FUNCTION FUNC_Bad : BOOL
VAR_INPUT
  nInput : INT;
END_VAR

FUNC_Bad := nInput > 0;

METHOD M_Helper : BOOL
M_Helper := TRUE;
END_METHOD

END_FUNCTION

(* stored: Version 1.1.0.1, ProductVersion 3.1.4024.12
   POU FUNC_Bad: Id {d1e2f3a4-b5c6-7890-abcd-ef1234567893}, SpecialFunc None
   Method M_Helper: Id {e1f2a3b4-c5d6-7890-abcd-ef1234567894} *)
